FUNCTION TFNumeroUltimi_N_TrasportiOccupati : UINT // Restituisce il numero di trasporti occupati, dall'ultimo all' n-esimo
VAR_INPUT
	//HandlingPackTable : POINTER TO TFHandlingPackTable;
	ArrayPacchi : POINTER TO DUT_ArrayPacchi; 					//Array contenente i pacchi sui trasporti				
	NTrasportiDaControllare : UINT;
END_VAR
VAR
	i : UINT;
END_VAR

TFNumeroUltimi_N_TrasportiOccupati := 0; 

//FOR i:= MAXDIMARRAYPACCHI TO (MAXDIMARRAYPACCHI - NTrasportiDaControllare - 1) BY -1 DO
FOR i:= 1 TO NTrasportiDaControllare DO
	IF i <= NTrasportiDaControllare AND NTrasportiDaControllare <= MAXDIMARRAYPACCHI THEN
		IF ArrayPacchi^.Pacco[i].ID.ID_Pacco[0] > 0 THEN
			TFNumeroUltimi_N_TrasportiOccupati := TFNumeroUltimi_N_TrasportiOccupati +1;
		END_IF
	ELSE
		RETURN;
	END_IF
END_FOR

END_FUNCTION

(* stored: Version 1.1.0.1, ProductVersion 3.1.4024.11
   POU TFNumeroUltimi_N_TrasportiOccupati: Id {8d6fdeef-7bd9-4211-9c1b-c0ea502d91bd}, SpecialFunc None *)
